// TIA Portal V19 export
FUNCTION "FC_EM_Feeding" : Void   // FC2, FBD
TITLE = Feeding
{ S7_Optimized_Access := 'TRUE' }
// stored: SetENOAutomatically false
BEGIN

REGION Network 1: ------------------------------------------------------------------------ Inputs ------------------------------------------------------------------------
END_REGION

REGION Network 2: Verwerking iFeedingSenCilOut
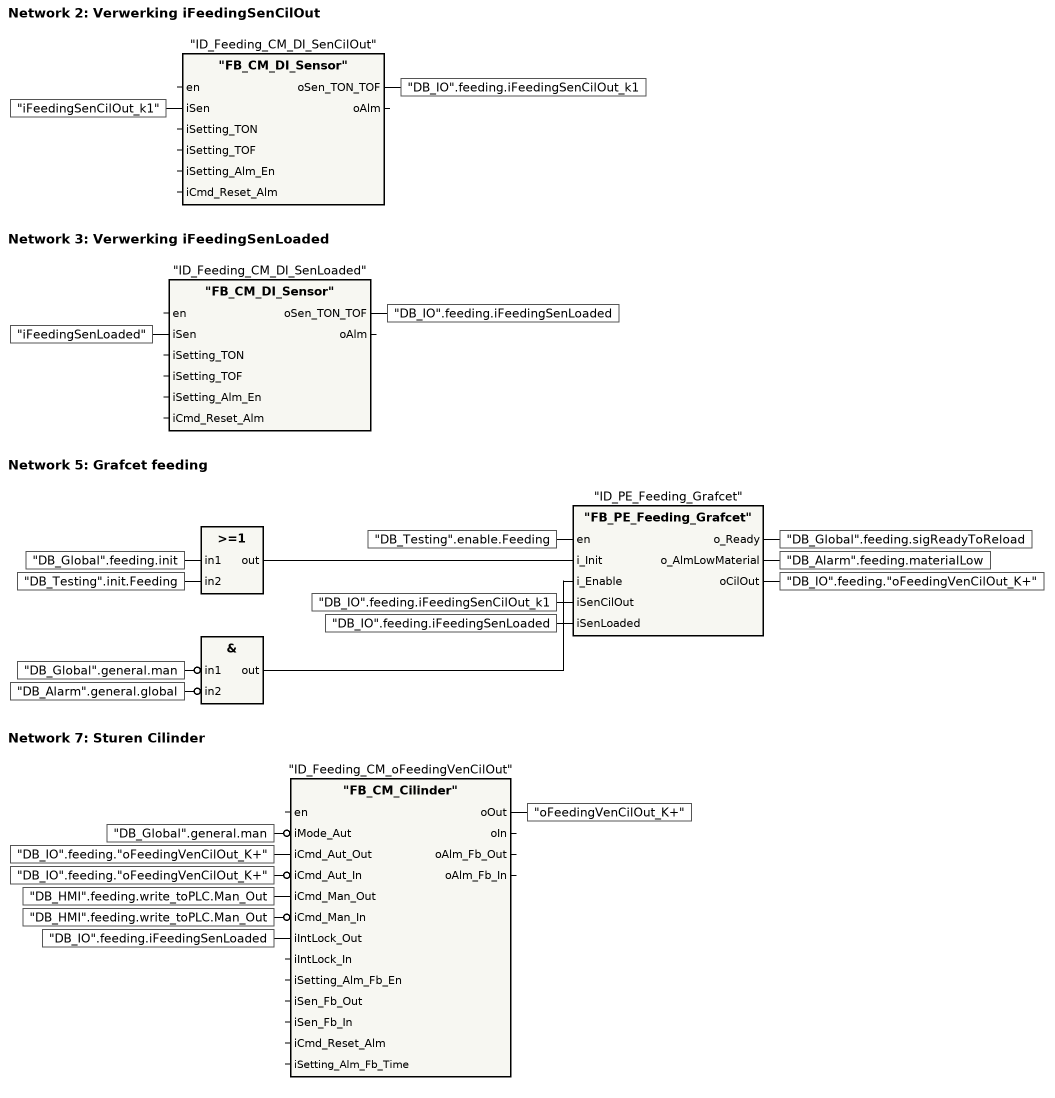
   "ID_Feeding_CM_DI_SenCilOut"(iSen := "iFeedingSenCilOut_k1",   // "FB_CM_DI_Sensor"
                           oSen_TON_TOF => "DB_IO".feeding.iFeedingSenCilOut_k1);
END_REGION

REGION Network 3: Verwerking iFeedingSenLoaded
   "ID_Feeding_CM_DI_SenLoaded"(iSen := "iFeedingSenLoaded", oSen_TON_TOF => "DB_IO".feeding.iFeedingSenLoaded);   // "FB_CM_DI_Sensor"
END_REGION

REGION Network 4: ------------------------------------------------------------------------ Logic ------------------------------------------------------------------------
END_REGION

REGION Network 5: Grafcet feeding
   IF "DB_Testing".enable.Feeding THEN
       "ID_PE_Feeding_Grafcet"(i_Init := "DB_Global".feeding.init OR "DB_Testing".init.Feeding,   // "FB_PE_Feeding_Grafcet"
                               i_Enable := NOT "DB_Global".general.man AND NOT "DB_Alarm".general.global,
                               iSenCilOut := "DB_IO".feeding.iFeedingSenCilOut_k1,
                               iSenLoaded := "DB_IO".feeding.iFeedingSenLoaded,
                               o_Ready => "DB_Global".feeding.sigReadyToReload,
                               o_AlmLowMaterial => "DB_Alarm".feeding.materialLow,
                               oCilOut => "DB_IO".feeding."oFeedingVenCilOut_K+");
   END_IF;
END_REGION

REGION Network 6: ------------------------------------------------------------------------ Outputs ------------------------------------------------------------------------
END_REGION

REGION Network 7: Sturen Cilinder
   "ID_Feeding_CM_oFeedingVenCilOut"(iMode_Aut := NOT "DB_Global".general.man,   // "FB_CM_Cilinder"
                           iCmd_Aut_Out := "DB_IO".feeding."oFeedingVenCilOut_K+",
                           iCmd_Aut_In := NOT "DB_IO".feeding."oFeedingVenCilOut_K+",
                           iCmd_Man_Out := "DB_HMI".feeding.write_toPLC.Man_Out,
                           iCmd_Man_In := NOT "DB_HMI".feeding.write_toPLC.Man_Out,
                           iIntLock_Out := "DB_IO".feeding.iFeedingSenLoaded,
                           oOut => "oFeedingVenCilOut_K+");
END_REGION
END_FUNCTION
